FUNCTION_BLOCK TEST_Skill EXTENDS FB_1_Skill
VAR_INPUT
END_VAR
VAR_OUTPUT
END_VAR
VAR
END_VAR

END_FUNCTION_BLOCK

(* stored: Version 1.1.0.1, ProductVersion 3.1.4026.18
   POU TEST_Skill: Id {fad47d1f-584c-43ef-9a86-749ff5c8ae2a}, SpecialFunc None *)
